FUNCTION_BLOCK EM_Doors EXTENDS EM_Base //??IMPLEMENTS I_EM_DOORS
VAR CONSTANT 
	c_nResultDataSize : UINT := 20;
END_VAR

VAR_INPUT
//Inputs
	i_stSettings : ST_SettingsDoors;
		
	i_bIlckOuterSpeedDoorToClose : BOOL; //TRUE = Interlocked
	i_bIlckOuterSpeedDoorToOpen : BOOL; //TRUE = Interlocked
	i_bIlckInnerSpeedDoorToClose : BOOL; //TRUE = Interlocked
	i_bIlckInnerSpeedDoorToOpen : BOOL; //TRUE = Interlocked
//++	i_bIlckCleanroomDoorToLock : BOOL; //TRUE = Interlocked
//++	i_bIlckCleanroomDoorToRelease : BOOL; //TRUE = Interlocked	

	i_ref_objCarrier : REFERENCE TO OBJ_Carrier;
END_VAR

VAR_OUTPUT
	q_bStaWarning : BOOL;
END_VAR

VAR
//------------------------------------------//
//Control Modules (Devices)
	s_cmOuterSpeedDoor : CM_SpeedDoor;
	s_cmInnerSpeedDoor : CM_SpeedDoor;	
//++	s_cmCleanroomDoor : CM_DoorLock;
//------------------------------------------//

//------------------------------------------//

	
	//..

//------------------------------------------//
//Outputs
	//..

//------------------------------------------//

//Requests
	s_bReqOpenOuterSpeedDoor : BOOL := FALSE;
	s_bReqCloseOuterSpeedDoor : BOOL := FALSE;
	s_bReqOpenInnerSpeedDoor : BOOL := FALSE;
	s_bReqCloseInnerSpeedDoor : BOOL := FALSE;
//++	s_bReqReleaseCleanroomDoor : BOOL := FALSE;
//++	s_bReqLockCleanroomDoor : BOOL := FALSE;
	
//Properties
	s_bStaOuterSpeedDoorOpened : BOOL := FALSE;
	s_bStaOuterSpeedDoorClosed : BOOL := FALSE;
	
	s_bStaInnerSpeedDoorOpened : BOOL := FALSE;
	s_bStaInnerSpeedDoorClosed : BOOL := FALSE;
	
//++	s_bStaCleanroomDoorOpened : BOOL := FALSE;
//++	s_bStaCleanroomDoorClosed : BOOL := FALSE;
//++	s_bStaCleanroomLockReleased : BOOL := FALSE;
//++	s_bStaCleanroomLockApplied : BOOL := FALSE;

//------------------------------------------//
//Params
//..
//------------------------------------------//

//------------------------------------------//
//Variables
	s_eSeqDoors : E_SeqDoors;
	s_fbSeqDoors : FB_SeqControl;
	
	// Interlocks
	s_bIlckOuterSpeedDoorToClose 			: BOOL := TRUE;
	s_bIlckOuterSpeedDoorToOpen		 		: BOOL := TRUE;
	
	s_bIlckInnerSpeedDoorToClose 			: BOOL := TRUE;
	s_bIlckInnerSpeedDoorToOpen		 		: BOOL := TRUE;
	
//++	s_bIlckCleanroomDoorToLock 			: BOOL := TRUE;
//++	s_bIlckCleanroomDoorToRelease		: BOOL := TRUE;
	
//------------------------------------------//

//------------------------------------------//

//------------------------------------------//
//Alarms
	s_bWrnOuterSpeedDoorNoAllowedToOpen : BOOL;
	s_bWrnOuterSpeedDoorNoAllowedToClose : BOOL;
	s_bWrnInnerSpeedDoorNoAllowedToOpen : BOOL;
	s_bWrnInnerSpeedDoorNoAllowedToClose : BOOL;
//++	s_bWrnCleanroomDoorNoAllowedToRelease : BOOL;
//++	s_bWrnCleanroomDoorNoAllowedToLock : BOOL;

	s_fbAlarmHandlerOuterSpeedDoorNoAllowedToOpen : FB_AlarmHandler;
	s_fbAlarmHandlerOuterSpeedDoorNoAllowedToClose : FB_AlarmHandler;
	s_fbAlarmHandlerInnerSpeedDoorNoAllowedToOpen : FB_AlarmHandler;
	s_fbAlarmHandlerInnerSpeedDoorNoAllowedToClose : FB_AlarmHandler;
//++	s_fbAlarmHandlerCleanroomDoorNoAllowedToRelease : FB_AlarmHandler;
//++	s_fbAlarmHandlerCleanroomDoorNoAllowedToLock : FB_AlarmHandler;
	
//------------------------------------------//

//------------------------------------------//
//Hmi
	s_fbHmiBtnReset						: FB_HmiBtn;
	
	s_fbHmiBtnCloseOuterSpeedDoor		: FB_HmiBtn;
	s_fbHmiBtnOpenOuterSpeedDoor		: FB_HmiBtn;
	
	s_fbHmiBtnCloseInnerSpeedDoor		: FB_HmiBtn;
	s_fbHmiBtnOpenInnerSpeedDoor		: FB_HmiBtn;
	
//++	s_fbHmiBtnApplyLockCleanroomDoor	: FB_HmiBtn;
//++	s_fbHmiBtnReleaseLockCleanroomDoor	: FB_HmiBtn;
	
	s_fbHmiLedOuterSpeedDoorClosed			: FB_HmiLed;
	s_fbHmiLedOuterSpeedDoorOpened			: FB_HmiLed;
	
	s_fbHmiLedInnerSpeedDoorClosed			: FB_HmiLed;
	s_fbHmiLedInnerSpeedDoorOpened			: FB_HmiLed;
	
//++	s_fbHmiLedCleanDoorClosed			: FB_HmiLed;
//++	s_fbHmiLedCleanDoorOpened			: FB_HmiLed;
//++	s_fbHmiLedCleanroomDoorLocked		: FB_HmiLed;
//++	s_fbHmiLedCleanroomDoorReleased		: FB_HmiLed;
	
//------------------------------------------//

	{warning '#TODO' Het zou beter zijn om dit onder te brengen in de onderstaande control modules}
	s_bHmiForceOutputEnabled : BOOL;
	s_bHmiForceOutputStartEnabled : BOOL;
END_VAR


SUPER^();

METHOD PROTECTED _m_Alarms : BOOL

IF NOT SUPER^._m_Alarms() THEN
	RETURN;
END_IF
	
	s_fbAlarmHandlerOuterSpeedDoorNoAllowedToOpen(
		i_bStaActive := i_bReqEnable AND s_bWrnOuterSpeedDoorNoAllowedToOpen,
		i_eAlarmLevel := E_AlarmLevel.Warning,
		i_sAlarmText := 'Outer Speed Door Not Allowed To Open');
	
	s_fbAlarmHandlerOuterSpeedDoorNoAllowedToClose(
		i_bStaActive := i_bReqEnable AND s_bWrnOuterSpeedDoorNoAllowedToClose,
		i_eAlarmLevel := E_AlarmLevel.Warning,
		i_sAlarmText := 'Outer Speed Door Not Allowed To Close');
		
	s_fbAlarmHandlerInnerSpeedDoorNoAllowedToOpen(
		i_bStaActive := i_bReqEnable AND s_bWrnInnerSpeedDoorNoAllowedToOpen,
		i_eAlarmLevel := E_AlarmLevel.Warning,
		i_sAlarmText := 'Inner Speed Door Not Allowed To Open');
	
	s_fbAlarmHandlerInnerSpeedDoorNoAllowedToClose(
		i_bStaActive := i_bReqEnable AND s_bWrnInnerSpeedDoorNoAllowedToClose,
		i_eAlarmLevel := E_AlarmLevel.Warning,
		i_sAlarmText := 'Inner Speed Door Not Allowed To Close');
	
//++	s_fbAlarmHandlerCleanroomDoorNoAllowedToRelease(
//++		i_bStaActive := i_bReqEnable AND s_bWrnCleanroomDoorNoAllowedToRelease,
//++		i_eAlarmLevel := E_AlarmLevel.Warning,
//++		i_sAlarmText := 'Cleanroom Door Not Allowed To Release/Open');
	
//++	s_fbAlarmHandlerCleanroomDoorNoAllowedToLock(
//++		i_bStaActive := i_bReqEnable AND s_bWrnCleanroomDoorNoAllowedToLock,
//++		i_eAlarmLevel := E_AlarmLevel.Warning,
//++		i_sAlarmText := 'Cleanroom Door Not Allowed To Lock');
	
	//Reset error/warning bits
	IF i_bCmdReset THEN
		s_bWrnOuterSpeedDoorNoAllowedToOpen := FALSE;
		s_bWrnOuterSpeedDoorNoAllowedToClose := FALSE;
		s_bWrnInnerSpeedDoorNoAllowedToOpen := FALSE;
		s_bWrnInnerSpeedDoorNoAllowedToClose := FALSE;
//++		s_bWrnCleanroomDoorNoAllowedToRelease := FALSE;
//++		s_bWrnCleanroomDoorNoAllowedToLock := FALSE;
	END_IF

_m_Alarms := TRUE;
END_METHOD

METHOD PROTECTED _m_Hmi : BOOL

IF NOT SUPER^._m_Hmi() THEN
	RETURN;
END_IF

//Buttons
s_fbHmiBtnReset();
	
s_fbHmiBtnCloseOuterSpeedDoor();
s_fbHmiBtnOpenOuterSpeedDoor();

s_fbHmiBtnCloseInnerSpeedDoor();
s_fbHmiBtnOpenInnerSpeedDoor();
	
//++s_fbHmiBtnApplyLockCleanroomDoor();;
//++s_fbHmiBtnReleaseLockCleanroomDoor();

//Leds	
s_fbHmiLedOuterSpeedDoorClosed(i_bStaLed := s_bStaOuterSpeedDoorClosed);
s_fbHmiLedOuterSpeedDoorOpened(i_bStaLed := s_bStaOuterSpeedDoorOpened);

s_fbHmiLedInnerSpeedDoorClosed(i_bStaLed := s_bStaInnerSpeedDoorClosed);
s_fbHmiLedInnerSpeedDoorOpened(i_bStaLed := s_bStaInnerSpeedDoorOpened);
	
//++s_fbHmiLedCleanDoorClosed(i_bStaLed := s_bStaCleanroomDoorClosed);
//++s_fbHmiLedCleanDoorOpened(i_bStaLed := s_bStaCleanroomDoorOpened);
//++s_fbHmiLedCleanroomDoorLocked(i_bStaLed := s_bStaCleanroomLockApplied);
//++s_fbHmiLedCleanroomDoorReleased(i_bStaLed := s_bStaCleanroomLockReleased);

_m_Hmi := TRUE;
END_METHOD

METHOD PROTECTED _m_Init : BOOL

IF NOT SUPER^._m_Init() THEN
	RETURN;
END_IF

//Interlock (externala + internal interlock reasons)
// Waarschijnlijk is het toch beter om de interlock uitsluited extern te verzamelen. Denk bijvoorbeeld aan de situatie dat er een box gedocked is (outer door is dan open), de claenroom deur mag in die sitiuatie geopende worden
s_bIlckOuterSpeedDoorToClose := i_bReqEnable AND i_bIlckOuterSpeedDoorToClose;
s_bIlckOuterSpeedDoorToOpen := i_bReqEnable AND i_bIlckOuterSpeedDoorToOpen;
s_bIlckInnerSpeedDoorToClose := i_bReqEnable AND i_bIlckInnerSpeedDoorToClose;
s_bIlckInnerSpeedDoorToOpen := i_bReqEnable AND i_bIlckInnerSpeedDoorToOpen;
//++s_bIlckCleanroomDoorToLock := i_bReqEnable AND i_bIlckCleanroomDoorToLock;
//++s_bIlckCleanroomDoorToRelease := i_bReqEnable AND i_bIlckCleanroomDoorToRelease;	

//Control Modules
s_cmOuterSpeedDoor.i_bReqEnable := FALSE;
s_cmOuterSpeedDoor.i_eCtrlMode := E_CtrlMode.IDLE;
s_cmOuterSpeedDoor.i_sCmName := 'Outer Speed Door';
s_cmOuterSpeedDoor.i_stSettings.tDoorClosingTimeout := T#10S;
s_cmOuterSpeedDoor.i_stSettings.tDoorOpeningTimeout := T#10S;
s_cmOuterSpeedDoor.i_stSettings.tResetPulseDuration := T#1S;
{warning '#TODO: Dot we need to added configuration parameters? Seperate struct or via settings or dedicateed variables'}

s_cmInnerSpeedDoor.i_bReqEnable := FALSE;
s_cmInnerSpeedDoor.i_eCtrlMode := E_CtrlMode.IDLE;
s_cmInnerSpeedDoor.i_sCmName := 'Inner Speed Door';
s_cmInnerSpeedDoor.i_stSettings.tDoorClosingTimeout := T#10S;
s_cmInnerSpeedDoor.i_stSettings.tDoorOpeningTimeout := T#10S;
s_cmInnerSpeedDoor.i_stSettings.tResetPulseDuration := T#1S;
{warning '#TODO: Dot we need to added configuration parameters? Seperate struct or via settings or dedicateed variables'}
	
//++s_cmCleanroomDoor.i_bReqEnable := FALSE;
//++s_cmCleanroomDoor.i_eCtrlMode := E_CtrlMode.IDLE;
//++s_cmCleanroomDoor.i_sCmName := 'Cleanroom Door';
//++s_cmCleanroomDoor.i_stSettings.tApplyingLockTimeout := T#3S;
//++s_cmCleanroomDoor.i_stSettings.tReleasingLockTimeout := T#3S;
//++{warning '#TODO: Dot we need to added configuration parameters? Seperate struct or via settings or dedicateed variables'}
	
//---------------------------------//	

//----------------------------------//

	
//----------------------------------//	
//Hmi
	s_fbHmiBtnReset.p_eButtontype := E_HmiButtonType.PUSHBUTTON;
	s_fbHmiBtnReset.p_bStaVisible := FALSE;
	s_fbHmiBtnReset.p_bStaEnabled := FALSE;		
	s_fbHmiBtnReset.p_sBtnText := 'Reset';
	
	s_fbHmiBtnCloseOuterSpeedDoor.p_eButtontype := E_HmiButtonType.PUSHBUTTON;
	s_fbHmiBtnCloseOuterSpeedDoor.p_bStaVisible := FALSE;
	s_fbHmiBtnCloseOuterSpeedDoor.p_bStaEnabled := FALSE;		
	s_fbHmiBtnCloseOuterSpeedDoor.p_sBtnText := 'Close Outer Speed Door';
	
	s_fbHmiBtnOpenOuterSpeedDoor.p_eButtontype := E_HmiButtonType.PUSHBUTTON;
	s_fbHmiBtnOpenOuterSpeedDoor.p_bStaVisible := FALSE;
	s_fbHmiBtnOpenOuterSpeedDoor.p_bStaEnabled := FALSE;		
	s_fbHmiBtnOpenOuterSpeedDoor.p_sBtnText := 'Open Outer Speed Door';
	
	s_fbHmiBtnCloseInnerSpeedDoor.p_eButtontype := E_HmiButtonType.PUSHBUTTON;
	s_fbHmiBtnCloseInnerSpeedDoor.p_bStaVisible := FALSE;
	s_fbHmiBtnCloseInnerSpeedDoor.p_bStaEnabled := FALSE;		
	s_fbHmiBtnCloseInnerSpeedDoor.p_sBtnText := 'Close Inner Speed Door';
	
	s_fbHmiBtnOpenInnerSpeedDoor.p_eButtontype := E_HmiButtonType.PUSHBUTTON;
	s_fbHmiBtnOpenInnerSpeedDoor.p_bStaVisible := FALSE;
	s_fbHmiBtnOpenInnerSpeedDoor.p_bStaEnabled := FALSE;		
	s_fbHmiBtnOpenInnerSpeedDoor.p_sBtnText := 'Open Inner Speed Door';
	
//++	s_fbHmiBtnApplyLockCleanroomDoor.p_eButtontype := E_HmiButtonType.PUSHBUTTON;
//++	s_fbHmiBtnApplyLockCleanroomDoor.p_bStaVisible := FALSE;
//++	s_fbHmiBtnApplyLockCleanroomDoor.p_bStaEnabled := FALSE;		
//++	s_fbHmiBtnApplyLockCleanroomDoor.p_sBtnText := 'Lock Cleanroom Door';
	
//++	s_fbHmiBtnReleaseLockCleanroomDoor.p_eButtontype := E_HmiButtonType.PUSHBUTTON;
//++	s_fbHmiBtnReleaseLockCleanroomDoor.p_bStaVisible := FALSE;
//++	s_fbHmiBtnReleaseLockCleanroomDoor.p_bStaEnabled := FALSE;		
//++	s_fbHmiBtnReleaseLockCleanroomDoor.p_sBtnText := 'Release Cleanroom Door';

	s_fbHmiLedOuterSpeedDoorClosed.p_bStaVisible := FALSE;
	s_fbHmiLedOuterSpeedDoorClosed.p_sToHmiDescriptionLed := 'Outer Speed Door Closed';
	
	s_fbHmiLedOuterSpeedDoorOpened.p_bStaVisible := FALSE;
	s_fbHmiLedOuterSpeedDoorOpened.p_sToHmiDescriptionLed := 'Outer Speed Door Opened';
	
	s_fbHmiLedInnerSpeedDoorClosed.p_bStaVisible := FALSE;
	s_fbHmiLedInnerSpeedDoorClosed.p_sToHmiDescriptionLed := 'Inner Speed Door Closed';
	
	s_fbHmiLedInnerSpeedDoorOpened.p_bStaVisible := FALSE;
	s_fbHmiLedInnerSpeedDoorOpened.p_sToHmiDescriptionLed := 'Inner Speed Door Opened';
	
//++	s_fbHmiLedCleanDoorClosed.p_bStaVisible := FALSE;
//++	s_fbHmiLedCleanDoorClosed.p_sToHmiDescriptionLed := 'Cleanroom Door Closed';
	
//++	s_fbHmiLedCleanDoorOpened.p_bStaVisible := FALSE;
//++	s_fbHmiLedCleanDoorOpened.p_sToHmiDescriptionLed := 'Cleanroom Door Opened';
	
//++	s_fbHmiLedCleanroomDoorLocked.p_bStaVisible := FALSE;
//++	s_fbHmiLedCleanroomDoorLocked.p_sToHmiDescriptionLed := 'Cleanroom Door Locked';
	
//++	s_fbHmiLedCleanroomDoorReleased.p_bStaVisible := FALSE;
//++	s_fbHmiLedCleanroomDoorReleased.p_sToHmiDescriptionLed := 'Cleanroom Door Released';
 
_m_Init := TRUE;
END_METHOD

METHOD PROTECTED _m_Inputs : BOOL

IF NOT SUPER^._m_Inputs() THEN
	RETURN;
END_IF


s_bIlckOuterSpeedDoorToOpen := i_bIlckOuterSpeedDoorToOpen;
s_bIlckOuterSpeedDoorToClose := i_bIlckOuterSpeedDoorToClose;

s_bIlckInnerSpeedDoorToOpen := i_bIlckInnerSpeedDoorToOpen;
s_bIlckInnerSpeedDoorToClose := i_bIlckInnerSpeedDoorToClose;
	
//++s_bIlckCleanroomDoorToRelease := i_bIlckCleanroomDoorToRelease;
//++s_bIlckCleanroomDoorToLock := i_bIlckCleanroomDoorToLock;

_m_Inputs := TRUE;
END_METHOD

METHOD PROTECTED _m_Modules : BOOL

IF NOT SUPER^._m_Devices() THEN
	RETURN;
END_IF

s_cmOuterSpeedDoor(
	i_bReqEnable := i_bReqEnable,
	i_eCtrlMode := i_eCtrlMode,
	i_bCmdReset := i_bCmdReset);

s_cmInnerSpeedDoor(
	i_bReqEnable := i_bReqEnable,
	i_eCtrlMode := i_eCtrlMode,
	i_bCmdReset := i_bCmdReset);
	
//++s_cmCleanroomDoor(
//++	i_bReqEnable := i_bReqEnable,
//++	i_eCtrlMode := i_eCtrlMode,
//++	i_bCmdReset := i_bCmdReset);

//Statusses
s_bStaOuterSpeedDoorClosed := s_cmOuterSpeedDoor.p_bStaIsClosed;
s_bStaOuterSpeedDoorOpened := s_cmOuterSpeedDoor.p_bStaIsOpened;

s_bStaInnerSpeedDoorClosed := s_cmInnerSpeedDoor.p_bStaIsClosed;
s_bStaInnerSpeedDoorOpened := s_cmInnerSpeedDoor.p_bStaIsOpened;

//++s_bStaCleanroomLockApplied := s_cmCleanroomDoor.p_bStaLockIsApplied;
//++s_bStaCleanroomLockReleased := s_cmCleanroomDoor.p_bStaLockIsReleased;
//++s_bStaCleanroomDoorClosed := s_cmCleanroomDoor.p_bStaDoorIsClosed;
//++s_bStaCleanroomDoorOpened := NOT(s_cmCleanroomDoor.p_bStaDoorIsClosed);

s_bStaError := s_cmOuterSpeedDoor.p_bStaError OR s_cmInnerSpeedDoor.p_bStaError; (* OR s_cmCleanroomDoor.p_bStaError;*)
	
_m_Modules := TRUE;
END_METHOD

METHOD PROTECTED _m_Outputs : BOOL

IF NOT SUPER^._m_Outputs() THEN
	RETURN;
END_IF

_m_Outputs := TRUE;
END_METHOD

METHOD PROTECTED _m_Params : BOOL

IF NOT SUPER^._m_Params() THEN
	RETURN;
END_IF

_m_Params := TRUE;
END_METHOD

METHOD PUBLIC m_ApplyLockCleanroomDoor : BOOL

IF NOT i_bReqEnable THEN 
	RETURN;
END_IF

IF NOT(FALSE) THEN
	s_bReqOpenOuterDoor := FALSE;
	s_bReqCloseOuterDoor := FALSE;
	s_bReqReleaseCleanroomDoor := FALSE;
	s_bReqLockCleanroomDoor := TRUE;
	
	m_ApplyLockCleanroomDoor := TRUE;
	
ELSE
	s_bWrnCleanroomDoorNoAllowedToLock := TRUE;
	
	m_ApplyLockCleanroomDoor := FALSE;
END_IF
END_METHOD

METHOD PUBLIC m_CloseInnerSpeedDoor : BOOL

IF NOT i_bReqEnable THEN 
	RETURN;
END_IF

IF NOT(s_bIlckInnerSpeedDoorToClose) THEN
	s_bReqOpenOuterSpeedDoor := FALSE;
	s_bReqCloseOuterSpeedDoor := FALSE;
	s_bReqOpenInnerSpeedDoor := FALSE;
	s_bReqCloseInnerSpeedDoor := TRUE;
//++	s_bReqReleaseCleanroomDoor := FALSE;
//++	s_bReqLockCleanroomDoor := FALSE;
	
	m_CloseInnerSpeedDoor := TRUE;
	
ELSE
	s_bWrnInnerSpeedDoorNoAllowedToClose := TRUE;
	
	m_CloseInnerSpeedDoor := FALSE;
END_IF
END_METHOD

METHOD PUBLIC m_CloseOuterSpeedDoor : BOOL

IF NOT i_bReqEnable THEN 
	RETURN;
END_IF

IF NOT(s_bIlckOuterSpeedDoorToClose) THEN
	s_bReqOpenOuterSpeedDoor := FALSE;
	s_bReqCloseOuterSpeedDoor := TRUE;
	s_bReqOpenInnerSpeedDoor := FALSE;
	s_bReqCloseInnerSpeedDoor := FALSE;
//++	s_bReqReleaseCleanroomDoor := FALSE;
//++	s_bReqLockCleanroomDoor := FALSE;
	
	m_CloseOuterSpeedDoor := TRUE;
	
ELSE
	s_bWrnOuterSpeedDoorNoAllowedToClose := TRUE;
	
	m_CloseOuterSpeedDoor := FALSE;
END_IF
END_METHOD

METHOD PUBLIC m_Main : BOOL

IF NOT SUPER^.m_Main() THEN
	RETURN;
END_IF

//Control of doors

{waring '#TODO: wrtie code below'}
(*

CASE i_eCtrlMode OF

	E_CtrlMode.IDLE:
		;
	
	E_CtrlMode.AUTOMATIC:
		
		CASE i_ref_objCarrier.p_eLocation OF 
	
			E_Location.PRE_DOCKING: //Control outer door
		
				IF i_ref_objCarrier.p_eDestination > E_Location.PRE_DOCKING THEN
					//Check if outer door is allowed to open
					IF NOT(i_bIlckOuterSpeedDoorToOpen) THEN
						s_cmOuterSpeedDoor();
					ELSE
						//Generate warning to user, door not allowed to open	
					END_IF
				END_IF
				
				IF p_bStaOuterSpeedDoorOpened THEN
					//Generate info to user, to place TB to docking position
				END_IF
				
				IF i_ref_objCarrier.p_eDestination <= E_Location.PRE_DOCKING THEN
					//Check if outer door is allowed to close
					IF NOT(i_bIlckOuterSpeedDoorToClose) THEN
						s_cmOuterSpeedDoor.m_Close();
					ELSE
						//Generate warning to user, door not allowed to close	
					END_IF
				END_IF
						
			E_Location.CLEAN_ROOM: //Control cleanroom door
		
				IF i_ref_objCarrier.p_eDestination >= E_Location.CLEAN_ROOM THEN
					//Check if cleanroom door lock is allowed to be released
					IF NOT(i_bIlckCleanroomDoorToRelease) THEN
						IF i_ref_objCarrier.p_bFlushedClean THEN
							s_cmCleanroomDoor.m_Release();
						ELSE
							//Generate warning to user, not flushed/clean
						END_IF		
					ELSE
						//Generate warning to user, door not allowed to be released	
					END_IF
				END_IF
				
				IF i_ref_objCarrier.p_eDestination <= E_Location.PRE_DOCKING THEN
					//Check if outer door is allowed to close
					IF NOT(i_bIlckCleanroomDoorToLock) THEN
						IF s_cmCleanroomDoor.p_bStaDoorIsClosed THEN
							s_cmCleanroomDoor.m_Apply();
						ELSE
							//Generate info to user, close cleanroom door
						END_IF	
					ELSE
						//Generate warning to user, door not allowed to lock	
					END_IF
				END_IF		
				
				
		END_CASE	
		
		
	
	E_CtrlMode.MANUAL:
		;
END_CASE

CASE i_eCtrlMode OF

	E_CtrlMode.IDLE:
		s_cmOuterSpeedDoor.m_Stop();
		s_cmCleanroomDoor.m_Apply();
		
	E_CtrlMode.AUTOMATIC:
		
		s_fbSeqDoors(
			i_nSeqStep := s_eSeqDoors, 
			i_sStepName := TO_STRING(s_fbSeqDoors.q_eActState), 
			i_bCmdReset := i_bCmdReset, 
			i_bStaError := s_bStaError);
	
		CASE s_eSeqDoors OF
			
			E_SeqDoors.IDLE:
				IF s_fbSeqDoors.q_bStaEntry THEN
					//Reset all requests
					s_bReqCloseOuterSpeedDoor := FALSE;
					s_bReqOpenOuterSpeedDoor := FALSE;
					s_bReqLockCleanroomDoor := FALSE;
					s_bReqReleaseCleanroomDoor := FALSE;
				END_IF
			
				//Requests from public mehtods (checked for interlocks)
				IF s_bReqCloseOuterSpeedDoor THEN
					s_eSeqDoors := E_SeqDoors.CLOSE_OUTER_DOOR;
					
				ELSIF s_bReqOpenOuterSpeedDoor THEN
					s_eSeqDoors := E_SeqDoors.OPEN_OUTER_DOOR;
					
				ELSIF s_bReqLockCleanroomDoor THEN
					s_eSeqDoors := E_SeqDoors.LOCK_CLEANROOM_DOOR;
					
				ELSIF s_bReqReleaseCleanroomDoor THEN
					s_eSeqDoors := E_SeqDoors.RELEASE_CLEANROOM_DOOR;
				END_IF
			
			E_SeqDoors.CLOSE_OUTER_DOOR:
				IF s_fbSeqDoors.q_bStaEntry THEN
					s_cmOuterSpeedDoor.m_Close();
				END_IF
				
				IF s_cmOuterSpeedDoor.p_bStaIsClosed THEN
					s_eSeqDoors := E_SeqDoors.OUTER_DOOR_CLOSED;
				ELSIF s_cmOuterSpeedDoor.p_bStaError THEN
					{warning '#TODO write add some info to error string'}
					s_eSeqDoors := E_SeqDoors.ERROR;
				ELSIF (s_fbSeqDoors.q_tmStepTime >= i_stSettings.tOuterDoorTimeout) THEN
					{warning '#TODO write add some info to error string'}
					s_eSeqDoors := E_SeqDoors.ERROR;	
				END_IF
			
			E_SeqDoors.OUTER_DOOR_CLOSED:
				s_eSeqDoors := E_SeqDoors.IDLE;	
			
			E_SeqDoors.OPEN_OUTER_DOOR:
				IF s_fbSeqDoors.q_bStaEntry THEN
					s_cmOuterSpeedDoor.m_Open();
				END_IF
				
				IF s_cmOuterSpeedDoor.p_bStaIsOpened THEN
					s_eSeqDoors := E_SeqDoors.OUTER_DOOR_OPENED;
				ELSIF s_cmOuterSpeedDoor.p_bStaError THEN
					{warning '#TODO write add some info to error string'}
					s_eSeqDoors := E_SeqDoors.ERROR;
				ELSIF (s_fbSeqDoors.q_tmStepTime >= i_stSettings.tOuterDoorTimeout) THEN
					{warning '#TODO write add some info to error string'}
					s_eSeqDoors := E_SeqDoors.ERROR;	
				END_IF
			
			E_SeqDoors.OUTER_DOOR_OPENED:
				s_eSeqDoors := E_SeqDoors.IDLE;
			
			E_SeqDoors.LOCK_CLEANROOM_DOOR:
				IF s_fbSeqDoors.q_bStaEntry THEN
					s_cmCleanroomDoor.m_Apply();
				END_IF
				
				IF s_cmCleanroomDoor.p_bStaLockIsApplied THEN
					s_eSeqDoors := E_SeqDoors.CLEANROOM_DOOR_LOCKED;
				ELSIF s_cmCleanroomDoor.p_bStaError THEN
					{warning '#TODO write add some info to error string'}
					s_eSeqDoors := E_SeqDoors.ERROR;
				ELSIF (s_fbSeqDoors.q_tmStepTime >= i_stSettings.tCleanroomDoorTimeout) THEN
					{warning '#TODO write add some info to error string'}
					s_eSeqDoors := E_SeqDoors.ERROR;	
				END_IF
			
			E_SeqDoors.CLEANROOM_DOOR_LOCKED:
				s_eSeqDoors := E_SeqDoors.IDLE;
						
			E_SeqDoors.RELEASE_CLEANROOM_DOOR:
				IF s_fbSeqDoors.q_bStaEntry THEN
					s_cmCleanroomDoor.m_Release();
				END_IF
				
				IF s_cmCleanroomDoor.p_bStaLockIsReleased THEN
					s_eSeqDoors := E_SeqDoors.CLEANROOM_DOOR_RELEASED;
				ELSIF s_cmCleanroomDoor.p_bStaError THEN
					{warning '#TODO write add some info to error string'}
					s_eSeqDoors := E_SeqDoors.ERROR;
				ELSIF (s_fbSeqDoors.q_tmStepTime >= i_stSettings.tCleanroomDoorTimeout) THEN
					{warning '#TODO write add some info to error string'}
					s_eSeqDoors := E_SeqDoors.ERROR;	
				END_IF
			
			E_SeqDoors.CLEANROOM_DOOR_RELEASED:
				s_eSeqDoors := E_SeqDoors.IDLE;
			
			E_SeqDockingInterface.READY:
				;
			
			E_SeqDockingInterface.ERROR:
				s_cmOuterSpeedDoor.m_Stop();
				s_cmCleanroomDoor.m_Apply();
			
				IF i_bCmdReset THEN
					//Reset errors (probebly alredy done in the methode devices)
					//--cmValveDockingClampsUpper.i_bCmdReset := TRUE;
				
					s_eSeqDoors := E_SeqDockingInterface.IDLE;
				END_IF
				
		END_CASE		
	
		
	E_CtrlMode.MANUAL:
		;
		{warning '#TODO: Add manual control from hmi'}

		// Outer Door
		IF s_fbHmiBtnOpenOuterSpeedDoor.p_osrBtnPress THEN
			s_cmOuterSpeedDoor.m_Open();
		ELSIF s_fbHmiBtnCloseOuterSpeedDoor.p_osrBtnPress THEN
			s_cmOuterSpeedDoor.m_Close();
		END_IF
		
		// Door Lock
		IF s_fbHmiBtnReleaseLockCleanroomDoor.p_osrBtnPress THEN
			s_cmCleanroomDoor.m_Release();
		ELSIF s_fbHmiBtnApplyLockCleanroomDoor.p_osrBtnPress THEN
			s_cmCleanroomDoor.m_Apply();
		END_IF
		
END_CASE
*)
END_METHOD

METHOD PUBLIC m_OpenInnerSpeedDoor : BOOL

IF NOT i_bReqEnable THEN 
	RETURN;
END_IF

IF NOT(s_bIlckInnerSpeedDoorToOpen) THEN
	s_bReqOpenOuterSpeedDoor := FALSE;
	s_bReqCloseOuterSpeedDoor := FALSE;
	s_bReqOpenInnerSpeedDoor := TRUE;
	s_bReqCloseInnerSpeedDoor := FALSE;
//++	s_bReqReleaseCleanroomDoor := FALSE;
//++	s_bReqLockCleanroomDoor := FALSE;
	
	m_OpenInnerSpeedDoor := TRUE;
ELSE
	
	s_bWrnInnerSpeedDoorNoAllowedToOpen := TRUE;
	
	m_OpenInnerSpeedDoor := FALSE;
END_IF
END_METHOD

METHOD PUBLIC m_OpenOuterSpeedDoor : BOOL

IF NOT i_bReqEnable THEN 
	RETURN;
END_IF

IF NOT(s_bIlckOuterSpeedDoorToOpen) THEN
	s_bReqOpenOuterSpeedDoor := TRUE;
	s_bReqCloseOuterSpeedDoor := FALSE;
	s_bReqOpenInnerSpeedDoor := FALSE;
	s_bReqCloseInnerSpeedDoor := FALSE;
//++	s_bReqReleaseCleanroomDoor := FALSE;
//++	s_bReqLockCleanroomDoor := FALSE;
	
	m_OpenOuterSpeedDoor := TRUE;
ELSE
	
	s_bWrnOuterSpeedDoorNoAllowedToOpen := TRUE;
	
	m_OpenOuterSpeedDoor := FALSE;
END_IF
END_METHOD

METHOD PUBLIC m_ReleaseLockCleanroomDoor : BOOL

IF NOT i_bReqEnable THEN 
	RETURN;
END_IF

IF NOT(s_bIlckCleanroomDoorToLock) THEN
	s_bReqOpenOuterDoor := FALSE;
	s_bReqCloseOuterDoor := FALSE;
	s_bReqReleaseCleanroomDoor := TRUE;
	s_bReqLockCleanroomDoor := FALSE;
	
	m_ReleaseLockCleanroomDoor := TRUE;
ELSE
	
	s_bWrnCleanroomDoorNoAllowedToRelease := TRUE;
	
	m_ReleaseLockCleanroomDoor := FALSE;
END_IF
END_METHOD

PROPERTY PUBLIC p_bStaCleanroomDoorClosed : BOOL
GET

p_bStaCleanroomDoorClosed := s_bStaCleanroomDoorClosed;
END_GET
END_PROPERTY

PROPERTY PUBLIC p_bStaCleanroomDoorOpened : BOOL
GET

p_bStaCleanroomDoorOpened := s_bStaCleanroomDoorOpened;
END_GET
END_PROPERTY

PROPERTY PUBLIC p_bStaCleanroomLockApplied : BOOL
GET

p_bStaCleanroomLockApplied := s_bStaCleanroomLockApplied;
END_GET
END_PROPERTY

PROPERTY PUBLIC p_bStaCleanroomLockReleased : BOOL
GET

p_bStaCleanroomLockReleased := s_bStaCleanroomLockReleased;
END_GET
END_PROPERTY

PROPERTY PUBLIC p_bStaInnerSpeedDoorClosed : BOOL
GET

p_bStaInnerSpeedDoorClosed := s_bStaInnerSpeedDoorClosed;
END_GET
END_PROPERTY

PROPERTY PUBLIC p_bStaInnerSpeedDoorOpened : BOOL
GET

p_bStaInnerSpeedDoorOpened := s_bStaInnerSpeedDoorOpened;
END_GET
END_PROPERTY

PROPERTY PUBLIC p_bStaOuterSpeedDoorClosed : BOOL
GET

p_bStaOuterSpeedDoorClosed := s_bStaOuterSpeedDoorClosed;
END_GET
END_PROPERTY

PROPERTY PUBLIC p_bStaOuterSpeedDoorOpened : BOOL
GET

p_bStaOuterSpeedDoorOpened := s_bStaOuterSpeedDoorOpened;
END_GET
END_PROPERTY

PROPERTY PUBLIC p_bStaReady : BOOL
GET

p_bStaReady := (s_eSeqDoors = E_SeqDoors.READY);
END_GET
END_PROPERTY

END_FUNCTION_BLOCK

(* stored: Version 1.1.0.1, ProductVersion 3.1.4024.12
   POU EM_Doors: Id {0ea26ddd-052a-4260-bfaf-0daade60103a}, SpecialFunc None
   Folder Base: Id {86d48589-7e2d-40d8-97de-3d4db9988d9a}
   Method _m_Alarms: Id {34703853-800b-4320-8e6c-49abce8785b7}
   Method _m_Hmi: Id {06e9697b-07d7-4e29-8455-791381b5d99d}
   Method _m_Init: Id {f5588ebd-495a-4c31-a7f5-23415377d40e}
   Method _m_Inputs: Id {08e3676c-19d2-4657-8762-4d7303d85c82}
   Method _m_Modules: Id {c18c3403-a619-4da8-8c16-d38b3f2bd5db}
   Method _m_Outputs: Id {f763b42e-2a14-49e4-aeec-3b4dc606af2b}
   Method _m_Params: Id {02936153-be53-403e-812d-8d9a77c13756}
   Method m_ApplyLockCleanroomDoor: Id {4499f858-1c66-4e87-af48-eca8a833d6ae}
   Method m_CloseInnerSpeedDoor: Id {8b9659e3-9892-4336-a3c2-49b887b841ee}
   Method m_CloseOuterSpeedDoor: Id {9c407a35-74a6-401d-8a18-b21be8c2d1a1}
   Method m_Main: Id {c1559ad6-cc3e-4059-9eff-299ddfbeac7b}
   Method m_OpenInnerSpeedDoor: Id {574f8d3a-fdc9-465e-913e-843f784f0e6e}
   Method m_OpenOuterSpeedDoor: Id {cacb32c9-2f39-45b3-a10f-fdd38f341162}
   Method m_ReleaseLockCleanroomDoor: Id {145de249-cc49-4a2e-a93a-16f786c2ecb4}
   Property p_bStaCleanroomDoorClosed: Id {3e867690-16e1-4e81-ad03-19ccedfb22c2}
   Get Get: Id {9548d166-8d83-4477-b001-d95261ddbc06}
   Property p_bStaCleanroomDoorOpened: Id {bb117a50-1725-4cdb-9157-fc2597312e4e}
   Get Get: Id {e91b025b-dae0-4ea7-97b1-57ee28a26a9b}
   Property p_bStaCleanroomLockApplied: Id {e6feb3e3-3717-426d-b652-dbbaa9ba0f43}
   Get Get: Id {0d6adf81-f180-40fd-b901-f0c227800da7}
   Property p_bStaCleanroomLockReleased: Id {a2b1d59d-5e34-4c2d-b724-72237d669c65}
   Get Get: Id {8ba433c5-2593-4dbc-a0e7-7b9acd8e39d7}
   Property p_bStaInnerSpeedDoorClosed: Id {e820ef87-a935-4e5a-9f4e-74f710eeaa35}
   Get Get: Id {723740c9-5feb-4d12-ae81-508dbaf06682}
   Property p_bStaInnerSpeedDoorOpened: Id {fd770672-09bf-4052-b33b-9e8aaacab69c}
   Get Get: Id {cd7d4a09-3f8f-4815-907b-09d35b18097b}
   Property p_bStaOuterSpeedDoorClosed: Id {e8474055-2ea6-4b59-a386-3fcee4ae9262}
   Get Get: Id {38689063-15e9-462f-9650-3e7d7a523f33}
   Property p_bStaOuterSpeedDoorOpened: Id {bc66e39f-ee2c-4f79-9694-10ac484efe5a}
   Get Get: Id {d7cea33e-5fa5-438f-8145-a6950abb53e6}
   Property p_bStaReady: Id {6d80e77c-9c68-4a12-b235-99de416ee985}
   Get Get: Id {ce2aa158-fba6-44ce-a41e-0f93cd362f98} *)
